% RSLogix 500 project AQUATIC CENTRE PLC UPGRADE - 21-11-05.RSS, saved by version 7.00.00.19 %
PROJECT "AQUATIC"    % processor: MicroLogix 1500 %

PROGRAM FILES
  LAD 2 "MAIN"  6 rungs
  LAD 3 "STATUS"  10 rungs
  LAD 4 "ALARMS"  24 rungs
  LAD 5 "SCREEN"  6 rungs

DATA FILES
  O0 OUTPUT  4 elements
  I1 INPUT  6 elements
  S2 STATUS  66 elements
  B3 BINARY  10 elements
  T4 TIMER  21 elements
  C5 COUNTER  1 elements
  R6 CONTROL  1 elements
  N7 INTEGER  32 elements
  F8 FLOAT  1 elements

LADDER 2 "MAIN"
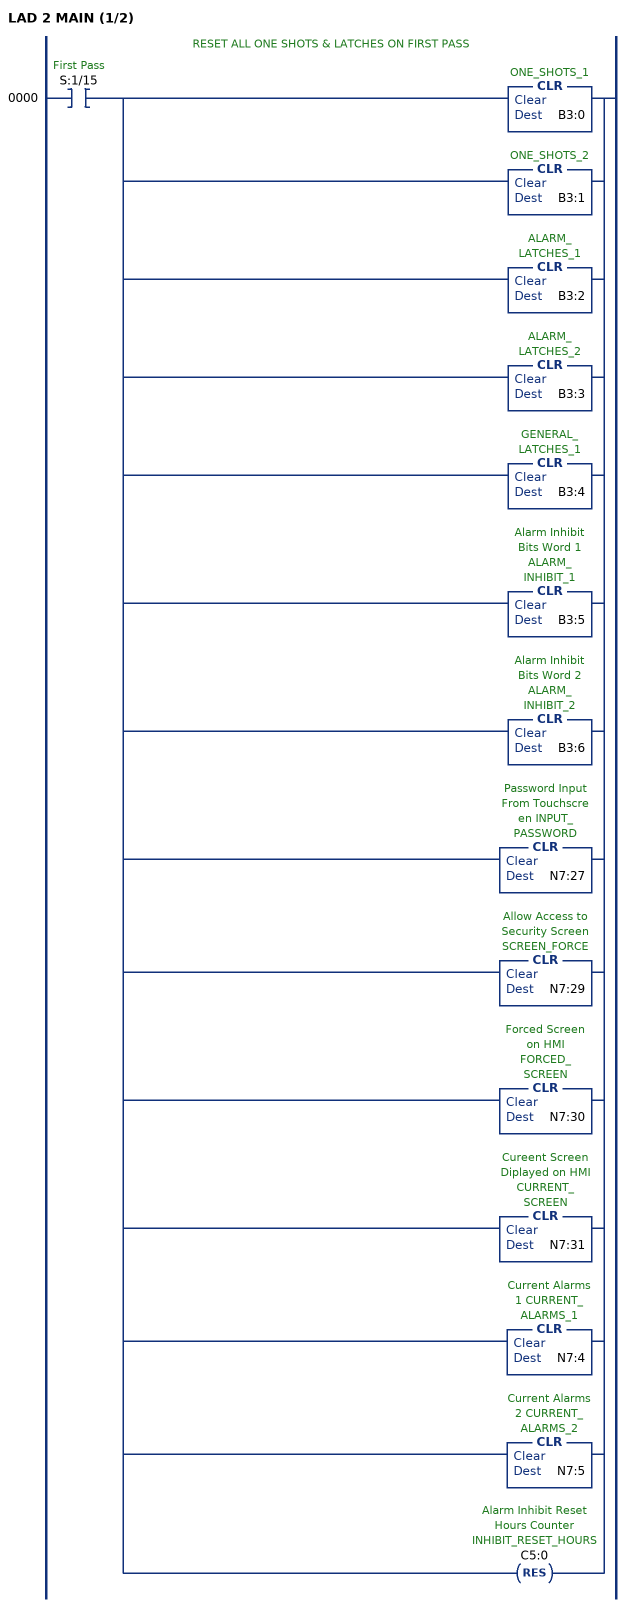
% Rung: 0 %
% RESET ALL ONE SHOTS & LATCHES ON FIRST PASS %
SOR XIC S:1/15 BST CLR B3:0 NXB CLR B3:1 NXB CLR B3:2 NXB CLR B3:3 NXB CLR B3:4 NXB CLR B3:5 NXB CLR B3:6 NXB CLR N7:27 NXB CLR N7:29 NXB CLR N7:30 NXB CLR N7:31 NXB CLR N7:4 NXB CLR N7:5 NXB RES C5:0 BND EOR
%   S:1/15  "First Pass" %
%   B3:0  ONE_SHOTS_1 %
%   B3:1  ONE_SHOTS_2 %
%   B3:2  ALARM_LATCHES_1 %
%   B3:3  ALARM_LATCHES_2 %
%   B3:4  GENERAL_LATCHES_1 %
%   B3:5  ALARM_INHIBIT_1  "Alarm Inhibit Bits Word 1" %
%   B3:6  ALARM_INHIBIT_2  "Alarm Inhibit Bits Word 2" %
%   N7:27  INPUT_PASSWORD  "Password Input From Touchscreen" %
%   N7:29  SCREEN_FORCE  "Allow Access to Security Screen" %
%   N7:30  FORCED_SCREEN  "Forced Screen on HMI" %
%   N7:31  CURRENT_SCREEN  "Cureent Screen Diplayed on HMI" %
%   N7:4  CURRENT_ALARMS_1  "Current Alarms 1" %
%   N7:5  CURRENT_ALARMS_2  "Current Alarms 2" %
%   C5:0  INHIBIT_RESET_HOURS  "Alarm Inhibit Reset Hours Counter" %

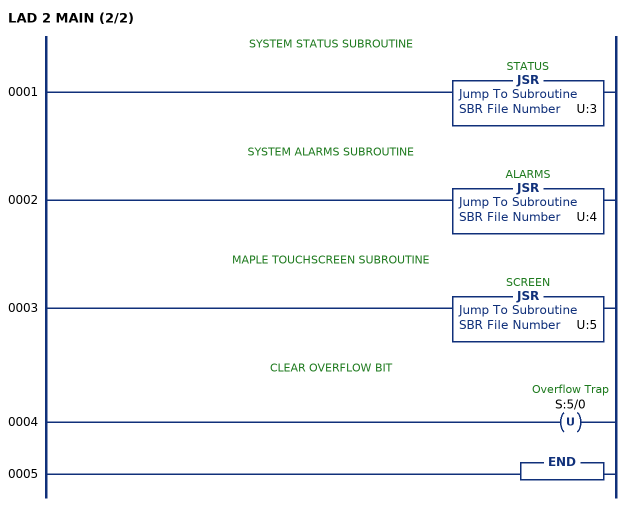
% Rung: 1 %
% SYSTEM STATUS SUBROUTINE %
SOR JSR U:3 EOR
%   U:3  STATUS %
% Rung: 2 %
% SYSTEM ALARMS SUBROUTINE %
SOR JSR U:4 EOR
%   U:4  ALARMS %
% Rung: 3 %
% MAPLE TOUCHSCREEN SUBROUTINE %
SOR JSR U:5 EOR
%   U:5  SCREEN %
% Rung: 4 %
% CLEAR OVERFLOW BIT %
SOR OTU S:5/0 EOR
%   S:5/0  "Overflow Trap" %
% Rung: 5 %
SOR END EOR

LADDER 3 "STATUS"
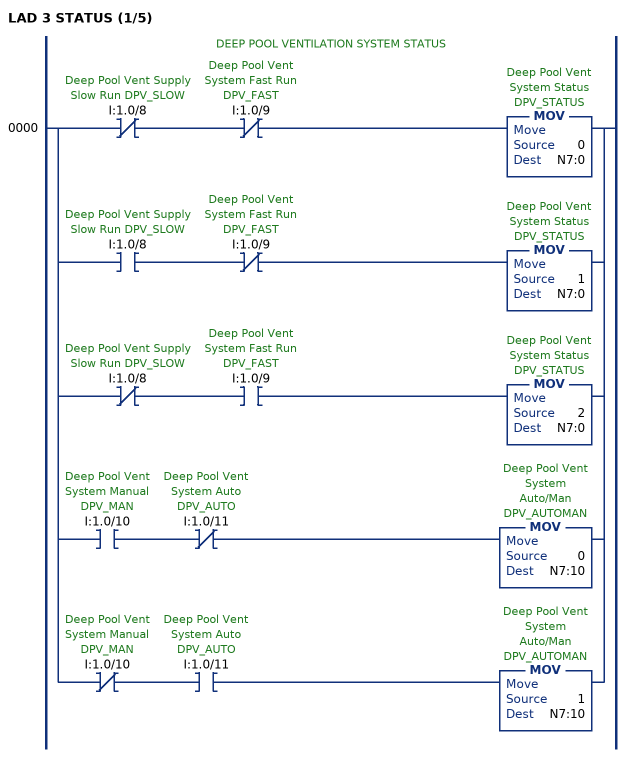
% Rung: 0 %
% DEEP POOL VENTILATION SYSTEM STATUS %
SOR BST XIO I:1.0/8 XIO I:1.0/9 MOV 0 N7:0 NXB XIC I:1.0/8 XIO I:1.0/9 MOV 1 N7:0 NXB XIO I:1.0/8 XIC I:1.0/9 MOV 2 N7:0 NXB XIC I:1.0/10 XIO I:1.0/11 MOV 0 N7:10 NXB XIO I:1.0/10 XIC I:1.0/11 MOV 1 N7:10 BND EOR
%   I:1.0/8  DPV_SLOW  "Deep Pool Vent Supply Slow Run" %
%   I:1.0/9  DPV_FAST  "Deep Pool Vent System Fast Run" %
%   N7:0  DPV_STATUS  "Deep Pool Vent System Status" %
%   I:1.0/10  DPV_MAN  "Deep Pool Vent System Manual" %
%   I:1.0/11  DPV_AUTO  "Deep Pool Vent System Auto" %
%   N7:10  DPV_AUTOMAN  "Deep Pool Vent System Auto/Man" %

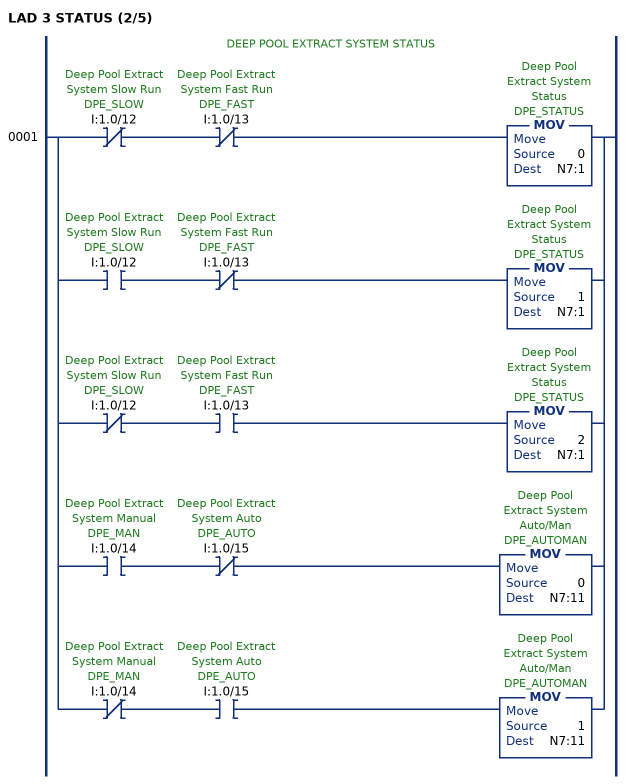
% Rung: 1 %
% DEEP POOL EXTRACT SYSTEM STATUS %
SOR BST XIO I:1.0/12 XIO I:1.0/13 MOV 0 N7:1 NXB XIC I:1.0/12 XIO I:1.0/13 MOV 1 N7:1 NXB XIO I:1.0/12 XIC I:1.0/13 MOV 2 N7:1 NXB XIC I:1.0/14 XIO I:1.0/15 MOV 0 N7:11 NXB XIO I:1.0/14 XIC I:1.0/15 MOV 1 N7:11 BND EOR
%   I:1.0/12  DPE_SLOW  "Deep Pool Extract System Slow Run" %
%   I:1.0/13  DPE_FAST  "Deep Pool Extract System Fast Run" %
%   N7:1  DPE_STATUS  "Deep Pool Extract System Status" %
%   I:1.0/14  DPE_MAN  "Deep Pool Extract System Manual" %
%   I:1.0/15  DPE_AUTO  "Deep Pool Extract System Auto" %
%   N7:11  DPE_AUTOMAN  "Deep Pool Extract System Auto/Man" %

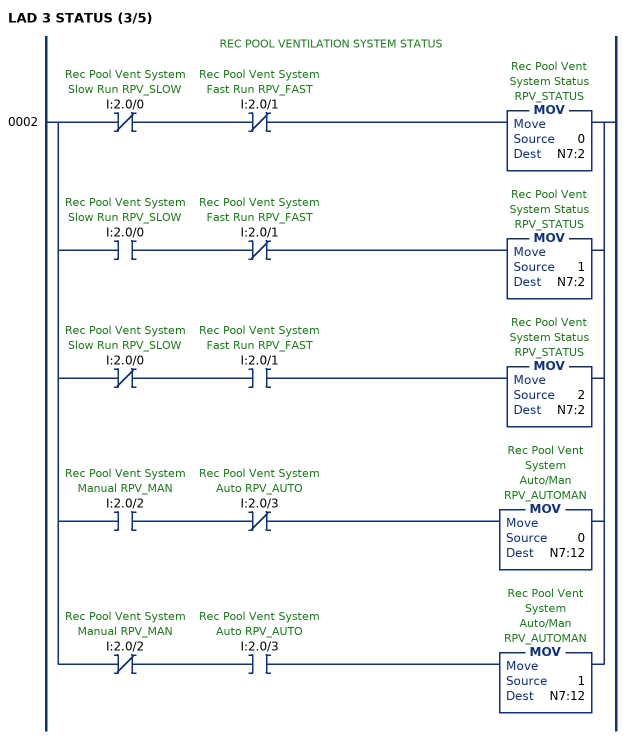
% Rung: 2 %
% REC POOL VENTILATION SYSTEM STATUS %
SOR BST XIO I:2.0/0 XIO I:2.0/1 MOV 0 N7:2 NXB XIC I:2.0/0 XIO I:2.0/1 MOV 1 N7:2 NXB XIO I:2.0/0 XIC I:2.0/1 MOV 2 N7:2 NXB XIC I:2.0/2 XIO I:2.0/3 MOV 0 N7:12 NXB XIO I:2.0/2 XIC I:2.0/3 MOV 1 N7:12 BND EOR
%   I:2.0/0  RPV_SLOW  "Rec Pool Vent System Slow Run" %
%   I:2.0/1  RPV_FAST  "Rec Pool Vent System Fast Run" %
%   N7:2  RPV_STATUS  "Rec Pool Vent System Status" %
%   I:2.0/2  RPV_MAN  "Rec Pool Vent System Manual" %
%   I:2.0/3  RPV_AUTO  "Rec Pool Vent System Auto" %
%   N7:12  RPV_AUTOMAN  "Rec Pool Vent System Auto/Man" %

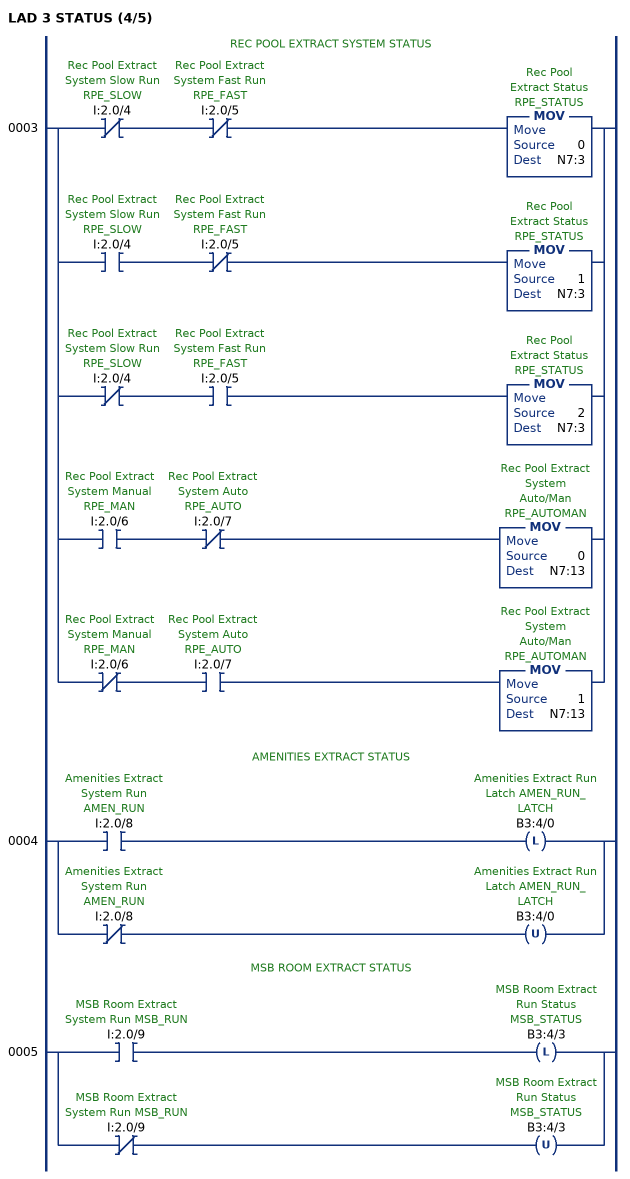
% Rung: 3 %
% REC POOL EXTRACT SYSTEM STATUS %
SOR BST XIO I:2.0/4 XIO I:2.0/5 MOV 0 N7:3 NXB XIC I:2.0/4 XIO I:2.0/5 MOV 1 N7:3 NXB XIO I:2.0/4 XIC I:2.0/5 MOV 2 N7:3 NXB XIC I:2.0/6 XIO I:2.0/7 MOV 0 N7:13 NXB XIO I:2.0/6 XIC I:2.0/7 MOV 1 N7:13 BND EOR
%   I:2.0/4  RPE_SLOW  "Rec Pool Extract System Slow Run" %
%   I:2.0/5  RPE_FAST  "Rec Pool Extract System Fast Run" %
%   N7:3  RPE_STATUS  "Rec Pool Extract Status" %
%   I:2.0/6  RPE_MAN  "Rec Pool Extract System Manual" %
%   I:2.0/7  RPE_AUTO  "Rec Pool Extract System Auto" %
%   N7:13  RPE_AUTOMAN  "Rec Pool Extract System Auto/Man" %
% Rung: 4 %
% AMENITIES EXTRACT STATUS %
SOR BST XIC I:2.0/8 OTL B3:4/0 NXB XIO I:2.0/8 OTU B3:4/0 BND EOR
%   I:2.0/8  AMEN_RUN  "Amenities Extract System Run" %
%   B3:4/0  AMEN_RUN_LATCH  "Amenities Extract Run Latch" %
% Rung: 5 %
% MSB ROOM EXTRACT STATUS %
SOR BST XIC I:2.0/9 OTL B3:4/3 NXB XIO I:2.0/9 OTU B3:4/3 BND EOR
%   I:2.0/9  MSB_RUN  "MSB Room Extract System Run" %
%   B3:4/3  MSB_STATUS  "MSB Room Extract Run Status" %

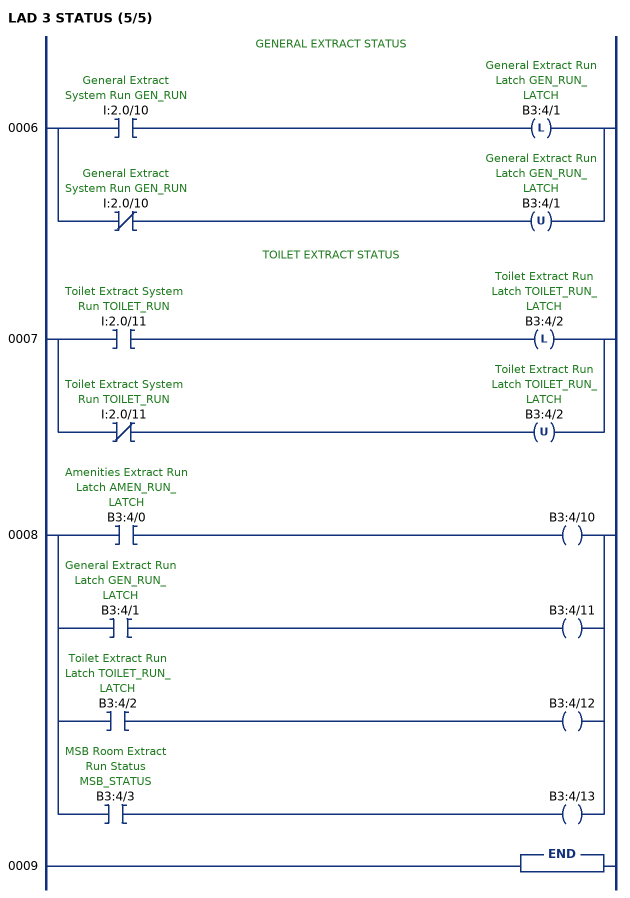
% Rung: 6 %
% GENERAL EXTRACT STATUS %
SOR BST XIC I:2.0/10 OTL B3:4/1 NXB XIO I:2.0/10 OTU B3:4/1 BND EOR
%   I:2.0/10  GEN_RUN  "General Extract System Run" %
%   B3:4/1  GEN_RUN_LATCH  "General Extract Run Latch" %
% Rung: 7 %
% TOILET EXTRACT STATUS %
SOR BST XIC I:2.0/11 OTL B3:4/2 NXB XIO I:2.0/11 OTU B3:4/2 BND EOR
%   I:2.0/11  TOILET_RUN  "Toilet Extract System Run" %
%   B3:4/2  TOILET_RUN_LATCH  "Toilet Extract Run Latch" %
% Rung: 8 %
SOR BST XIC B3:4/0 OTE B3:4/10 NXB XIC B3:4/1 OTE B3:4/11 NXB XIC B3:4/2 OTE B3:4/12 NXB XIC B3:4/3 OTE B3:4/13 BND EOR
%   B3:4/0  AMEN_RUN_LATCH  "Amenities Extract Run Latch" %
%   B3:4/1  GEN_RUN_LATCH  "General Extract Run Latch" %
%   B3:4/2  TOILET_RUN_LATCH  "Toilet Extract Run Latch" %
%   B3:4/3  MSB_STATUS  "MSB Room Extract Run Status" %
% Rung: 9 %
SOR END EOR

LADDER 4 "ALARMS"
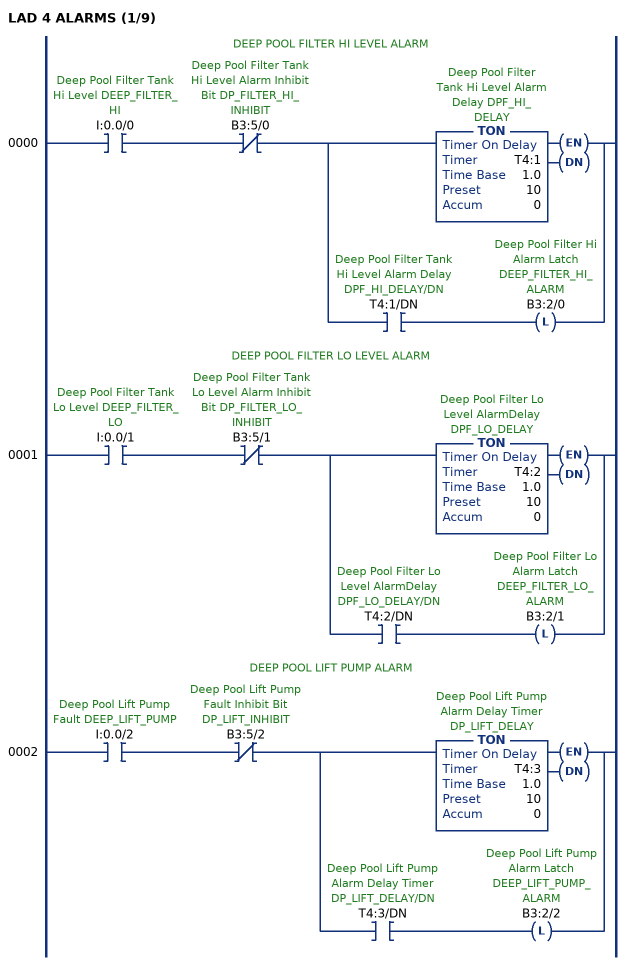
% Rung: 0 %
% DEEP POOL FILTER HI LEVEL ALARM %
SOR XIC I:0.0/0 XIO B3:5/0 BST TON T4:1 1.0 10 0 NXB XIC T4:1/DN OTL B3:2/0 BND EOR
%   I:0.0/0  DEEP_FILTER_HI  "Deep Pool Filter Tank Hi Level" %
%   B3:5/0  DP_FILTER_HI_INHIBIT  "Deep Pool Filter Tank Hi Level Alarm Inhibit Bit" %
%   T4:1  DPF_HI_DELAY  "Deep Pool Filter Tank Hi Level Alarm Delay" %
%   B3:2/0  DEEP_FILTER_HI_ALARM  "Deep Pool Filter Hi Alarm Latch" %
% Rung: 1 %
% DEEP POOL FILTER LO LEVEL ALARM %
SOR XIC I:0.0/1 XIO B3:5/1 BST TON T4:2 1.0 10 0 NXB XIC T4:2/DN OTL B3:2/1 BND EOR
%   I:0.0/1  DEEP_FILTER_LO  "Deep Pool Filter Tank Lo Level" %
%   B3:5/1  DP_FILTER_LO_INHIBIT  "Deep Pool Filter Tank Lo Level Alarm Inhibit Bit" %
%   T4:2  DPF_LO_DELAY  "Deep Pool Filter Lo Level AlarmDelay" %
%   B3:2/1  DEEP_FILTER_LO_ALARM  "Deep Pool Filter Lo Alarm Latch" %
% Rung: 2 %
% DEEP POOL LIFT PUMP ALARM %
SOR XIC I:0.0/2 XIO B3:5/2 BST TON T4:3 1.0 10 0 NXB XIC T4:3/DN OTL B3:2/2 BND EOR
%   I:0.0/2  DEEP_LIFT_PUMP  "Deep Pool Lift Pump Fault" %
%   B3:5/2  DP_LIFT_INHIBIT  "Deep Pool Lift Pump Fault Inhibit Bit" %
%   T4:3  DP_LIFT_DELAY  "Deep Pool Lift Pump Alarm Delay Timer" %
%   B3:2/2  DEEP_LIFT_PUMP_ALARM  "Deep Pool Lift Pump Alarm Latch" %

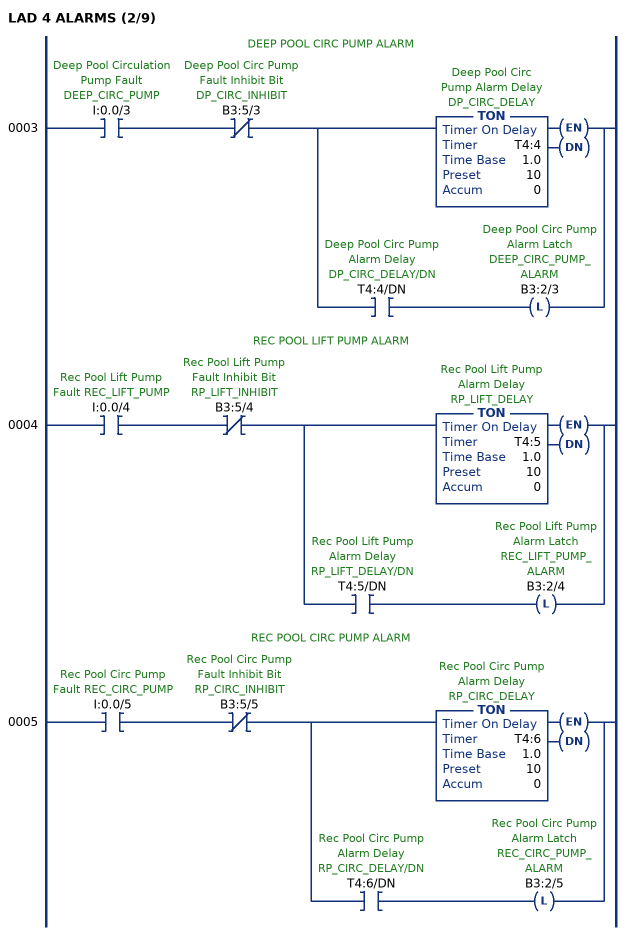
% Rung: 3 %
% DEEP POOL CIRC PUMP ALARM %
SOR XIC I:0.0/3 XIO B3:5/3 BST TON T4:4 1.0 10 0 NXB XIC T4:4/DN OTL B3:2/3 BND EOR
%   I:0.0/3  DEEP_CIRC_PUMP  "Deep Pool Circulation Pump Fault" %
%   B3:5/3  DP_CIRC_INHIBIT  "Deep Pool Circ Pump Fault Inhibit Bit" %
%   T4:4  DP_CIRC_DELAY  "Deep Pool Circ Pump Alarm Delay" %
%   B3:2/3  DEEP_CIRC_PUMP_ALARM  "Deep Pool Circ Pump Alarm Latch" %
% Rung: 4 %
% REC POOL LIFT PUMP ALARM %
SOR XIC I:0.0/4 XIO B3:5/4 BST TON T4:5 1.0 10 0 NXB XIC T4:5/DN OTL B3:2/4 BND EOR
%   I:0.0/4  REC_LIFT_PUMP  "Rec Pool Lift Pump Fault" %
%   B3:5/4  RP_LIFT_INHIBIT  "Rec Pool Lift Pump Fault Inhibit Bit" %
%   T4:5  RP_LIFT_DELAY  "Rec Pool Lift Pump Alarm Delay" %
%   B3:2/4  REC_LIFT_PUMP_ALARM  "Rec Pool Lift Pump Alarm Latch" %
% Rung: 5 %
% REC POOL CIRC PUMP ALARM %
SOR XIC I:0.0/5 XIO B3:5/5 BST TON T4:6 1.0 10 0 NXB XIC T4:6/DN OTL B3:2/5 BND EOR
%   I:0.0/5  REC_CIRC_PUMP  "Rec Pool Circ Pump Fault" %
%   B3:5/5  RP_CIRC_INHIBIT  "Rec Pool Circ Pump Fault Inhibit Bit" %
%   T4:6  RP_CIRC_DELAY  "Rec Pool Circ Pump Alarm Delay" %
%   B3:2/5  REC_CIRC_PUMP_ALARM  "Rec Pool Circ Pump Alarm Latch" %

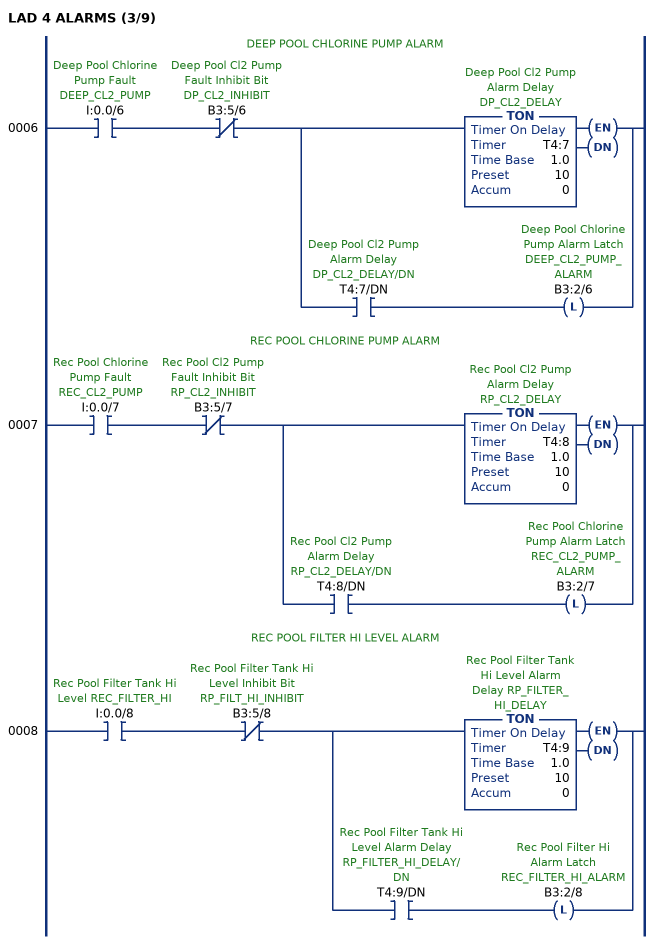
% Rung: 6 %
% DEEP POOL CHLORINE PUMP ALARM %
SOR XIC I:0.0/6 XIO B3:5/6 BST TON T4:7 1.0 10 0 NXB XIC T4:7/DN OTL B3:2/6 BND EOR
%   I:0.0/6  DEEP_CL2_PUMP  "Deep Pool Chlorine Pump Fault" %
%   B3:5/6  DP_CL2_INHIBIT  "Deep Pool Cl2 Pump Fault Inhibit Bit" %
%   T4:7  DP_CL2_DELAY  "Deep Pool Cl2 Pump Alarm Delay" %
%   B3:2/6  DEEP_CL2_PUMP_ALARM  "Deep Pool Chlorine Pump Alarm Latch" %
% Rung: 7 %
% REC POOL CHLORINE PUMP ALARM %
SOR XIC I:0.0/7 XIO B3:5/7 BST TON T4:8 1.0 10 0 NXB XIC T4:8/DN OTL B3:2/7 BND EOR
%   I:0.0/7  REC_CL2_PUMP  "Rec Pool Chlorine Pump Fault" %
%   B3:5/7  RP_CL2_INHIBIT  "Rec Pool Cl2 Pump Fault Inhibit Bit" %
%   T4:8  RP_CL2_DELAY  "Rec Pool Cl2 Pump Alarm Delay" %
%   B3:2/7  REC_CL2_PUMP_ALARM  "Rec Pool Chlorine Pump Alarm Latch" %
% Rung: 8 %
% REC POOL FILTER HI LEVEL ALARM %
SOR XIC I:0.0/8 XIO B3:5/8 BST TON T4:9 1.0 10 0 NXB XIC T4:9/DN OTL B3:2/8 BND EOR
%   I:0.0/8  REC_FILTER_HI  "Rec Pool Filter Tank Hi Level" %
%   B3:5/8  RP_FILT_HI_INHIBIT  "Rec Pool Filter Tank Hi Level Inhibit Bit" %
%   T4:9  RP_FILTER_HI_DELAY  "Rec Pool Filter Tank Hi Level Alarm Delay" %
%   B3:2/8  REC_FILTER_HI_ALARM  "Rec Pool Filter Hi Alarm Latch" %

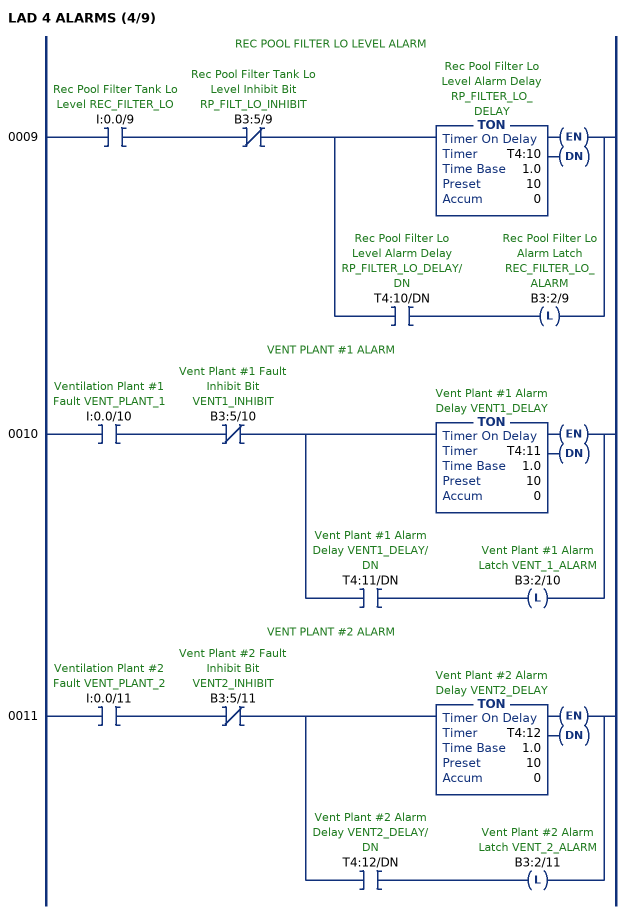
% Rung: 9 %
% REC POOL FILTER LO LEVEL ALARM %
SOR XIC I:0.0/9 XIO B3:5/9 BST TON T4:10 1.0 10 0 NXB XIC T4:10/DN OTL B3:2/9 BND EOR
%   I:0.0/9  REC_FILTER_LO  "Rec Pool Filter Tank Lo Level" %
%   B3:5/9  RP_FILT_LO_INHIBIT  "Rec Pool Filter Tank Lo Level Inhibit Bit" %
%   T4:10  RP_FILTER_LO_DELAY  "Rec Pool Filter Lo Level Alarm Delay" %
%   B3:2/9  REC_FILTER_LO_ALARM  "Rec Pool Filter Lo Alarm Latch" %
% Rung: 10 %
% VENT PLANT #1 ALARM %
SOR XIC I:0.0/10 XIO B3:5/10 BST TON T4:11 1.0 10 0 NXB XIC T4:11/DN OTL B3:2/10 BND EOR
%   I:0.0/10  VENT_PLANT_1  "Ventilation Plant #1 Fault" %
%   B3:5/10  VENT1_INHIBIT  "Vent Plant #1 Fault Inhibit Bit" %
%   T4:11  VENT1_DELAY  "Vent Plant #1 Alarm Delay" %
%   B3:2/10  VENT_1_ALARM  "Vent Plant #1 Alarm Latch" %
% Rung: 11 %
% VENT PLANT #2 ALARM %
SOR XIC I:0.0/11 XIO B3:5/11 BST TON T4:12 1.0 10 0 NXB XIC T4:12/DN OTL B3:2/11 BND EOR
%   I:0.0/11  VENT_PLANT_2  "Ventilation Plant #2 Fault" %
%   B3:5/11  VENT2_INHIBIT  "Vent Plant #2 Fault Inhibit Bit" %
%   T4:12  VENT2_DELAY  "Vent Plant #2 Alarm Delay" %
%   B3:2/11  VENT_2_ALARM  "Vent Plant #2 Alarm Latch" %

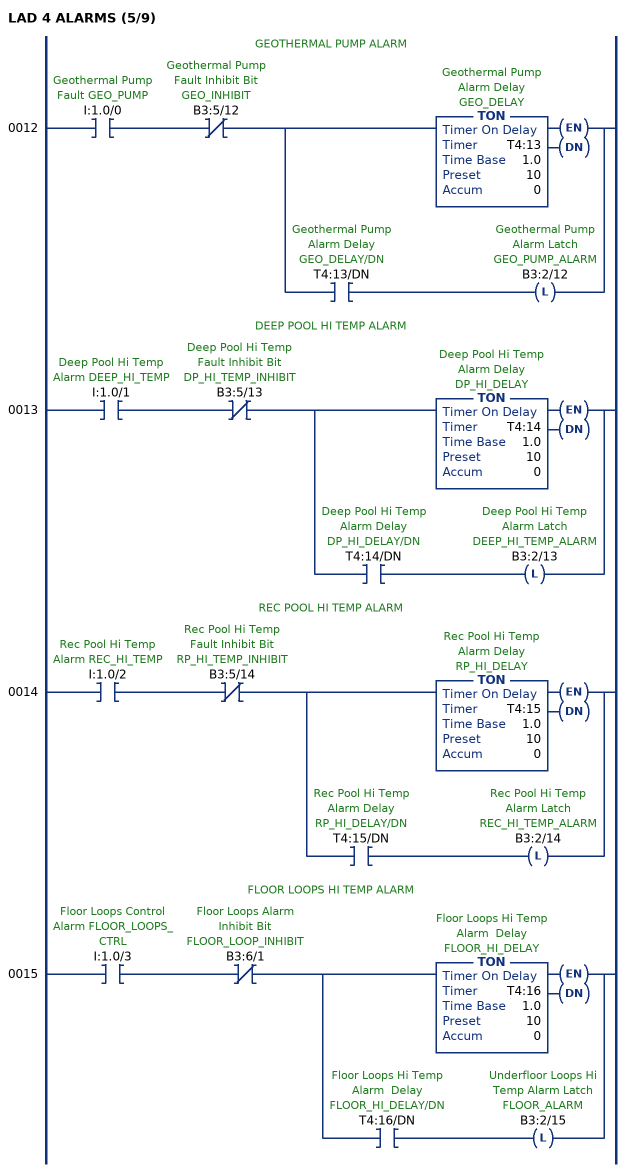
% Rung: 12 %
% GEOTHERMAL PUMP ALARM %
SOR XIC I:1.0/0 XIO B3:5/12 BST TON T4:13 1.0 10 0 NXB XIC T4:13/DN OTL B3:2/12 BND EOR
%   I:1.0/0  GEO_PUMP  "Geothermal Pump Fault" %
%   B3:5/12  GEO_INHIBIT  "Geothermal Pump Fault Inhibit Bit" %
%   T4:13  GEO_DELAY  "Geothermal Pump Alarm Delay" %
%   B3:2/12  GEO_PUMP_ALARM  "Geothermal Pump Alarm Latch" %
% Rung: 13 %
% DEEP POOL HI TEMP ALARM %
SOR XIC I:1.0/1 XIO B3:5/13 BST TON T4:14 1.0 10 0 NXB XIC T4:14/DN OTL B3:2/13 BND EOR
%   I:1.0/1  DEEP_HI_TEMP  "Deep Pool Hi Temp Alarm" %
%   B3:5/13  DP_HI_TEMP_INHIBIT  "Deep Pool Hi Temp Fault Inhibit Bit" %
%   T4:14  DP_HI_DELAY  "Deep Pool Hi Temp Alarm Delay" %
%   B3:2/13  DEEP_HI_TEMP_ALARM  "Deep Pool Hi Temp Alarm Latch" %
% Rung: 14 %
% REC POOL HI TEMP ALARM %
SOR XIC I:1.0/2 XIO B3:5/14 BST TON T4:15 1.0 10 0 NXB XIC T4:15/DN OTL B3:2/14 BND EOR
%   I:1.0/2  REC_HI_TEMP  "Rec Pool Hi Temp Alarm" %
%   B3:5/14  RP_HI_TEMP_INHIBIT  "Rec Pool Hi Temp Fault Inhibit Bit" %
%   T4:15  RP_HI_DELAY  "Rec Pool Hi Temp Alarm Delay" %
%   B3:2/14  REC_HI_TEMP_ALARM  "Rec Pool Hi Temp Alarm Latch" %
% Rung: 15 %
% FLOOR LOOPS HI TEMP ALARM %
SOR XIC I:1.0/3 XIO B3:6/1 BST TON T4:16 1.0 10 0 NXB XIC T4:16/DN OTL B3:2/15 BND EOR
%   I:1.0/3  FLOOR_LOOPS_CTRL  "Floor Loops Control Alarm" %
%   B3:6/1  FLOOR_LOOP_INHIBIT  "Floor Loops Alarm Inhibit Bit" %
%   T4:16  FLOOR_HI_DELAY  "Floor Loops Hi Temp Alarm  Delay" %
%   B3:2/15  FLOOR_ALARM  "Underfloor Loops Hi Temp Alarm Latch" %

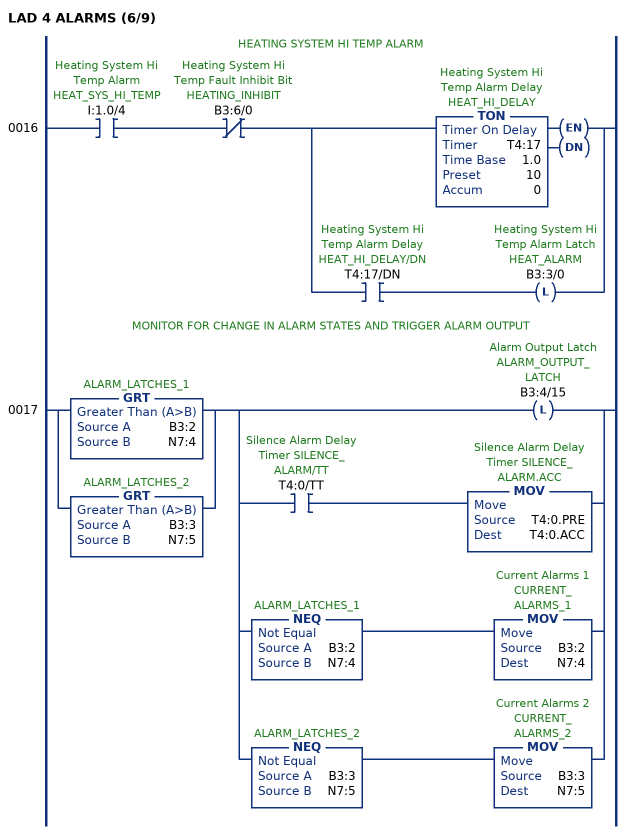
% Rung: 16 %
% HEATING SYSTEM HI TEMP ALARM %
SOR XIC I:1.0/4 XIO B3:6/0 BST TON T4:17 1.0 10 0 NXB XIC T4:17/DN OTL B3:3/0 BND EOR
%   I:1.0/4  HEAT_SYS_HI_TEMP  "Heating System Hi Temp Alarm" %
%   B3:6/0  HEATING_INHIBIT  "Heating System Hi Temp Fault Inhibit Bit" %
%   T4:17  HEAT_HI_DELAY  "Heating System Hi Temp Alarm Delay" %
%   B3:3/0  HEAT_ALARM  "Heating System Hi Temp Alarm Latch" %
% Rung: 17 %
% MONITOR FOR CHANGE IN ALARM STATES AND TRIGGER ALARM OUTPUT %
SOR BST GRT B3:2 N7:4 NXB GRT B3:3 N7:5 BND BST OTL B3:4/15 NXB XIC T4:0/TT MOV T4:0.PRE T4:0.ACC NXB NEQ B3:2 N7:4 MOV B3:2 N7:4 NXB NEQ B3:3 N7:5 MOV B3:3 N7:5 BND EOR
%   B3:2  ALARM_LATCHES_1 %
%   N7:4  CURRENT_ALARMS_1  "Current Alarms 1" %
%   B3:3  ALARM_LATCHES_2 %
%   N7:5  CURRENT_ALARMS_2  "Current Alarms 2" %
%   B3:4/15  ALARM_OUTPUT_LATCH  "Alarm Output Latch" %
%   T4:0  SILENCE_ALARM  "Silence Alarm Delay Timer" %

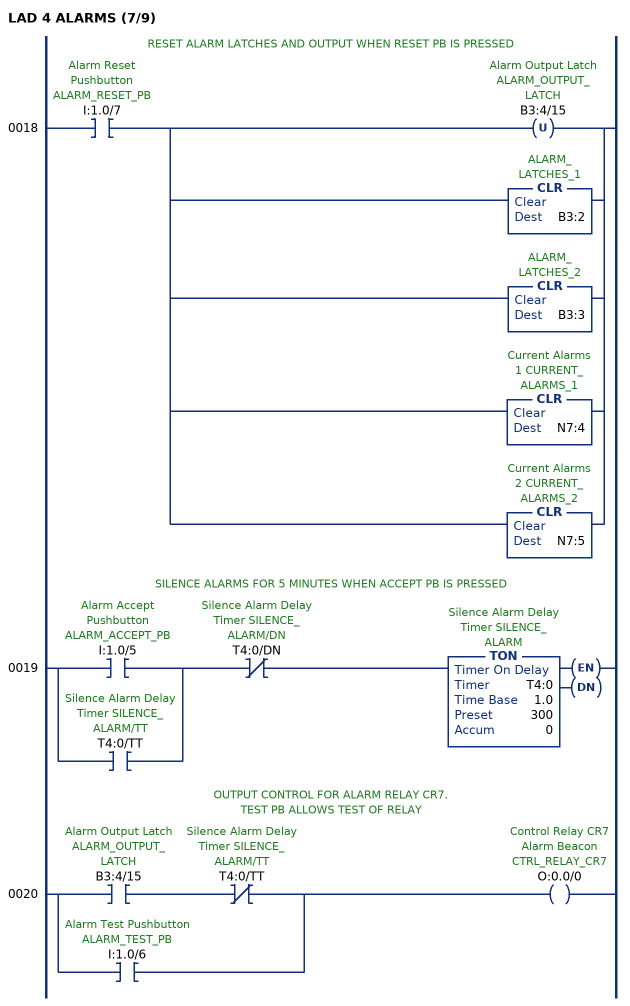
% Rung: 18 %
% RESET ALARM LATCHES AND OUTPUT WHEN RESET PB IS PRESSED %
SOR XIC I:1.0/7 BST OTU B3:4/15 NXB CLR B3:2 NXB CLR B3:3 NXB CLR N7:4 NXB CLR N7:5 BND EOR
%   I:1.0/7  ALARM_RESET_PB  "Alarm Reset Pushbutton" %
%   B3:4/15  ALARM_OUTPUT_LATCH  "Alarm Output Latch" %
%   B3:2  ALARM_LATCHES_1 %
%   B3:3  ALARM_LATCHES_2 %
%   N7:4  CURRENT_ALARMS_1  "Current Alarms 1" %
%   N7:5  CURRENT_ALARMS_2  "Current Alarms 2" %
% Rung: 19 %
% SILENCE ALARMS FOR 5 MINUTES WHEN ACCEPT PB IS PRESSED %
SOR BST XIC I:1.0/5 NXB XIC T4:0/TT BND XIO T4:0/DN TON T4:0 1.0 300 0 EOR
%   I:1.0/5  ALARM_ACCEPT_PB  "Alarm Accept Pushbutton" %
%   T4:0  SILENCE_ALARM  "Silence Alarm Delay Timer" %
% Rung: 20 %
% OUTPUT CONTROL FOR ALARM RELAY CR7.
% TEST PB ALLOWS TEST OF RELAY %
SOR BST XIC B3:4/15 XIO T4:0/TT NXB XIC I:1.0/6 BND OTE O:0.0/0 EOR
%   B3:4/15  ALARM_OUTPUT_LATCH  "Alarm Output Latch" %
%   T4:0  SILENCE_ALARM  "Silence Alarm Delay Timer" %
%   I:1.0/6  ALARM_TEST_PB  "Alarm Test Pushbutton" %
%   O:0.0/0  CTRL_RELAY_CR7  "Control Relay CR7 Alarm Beacon" %

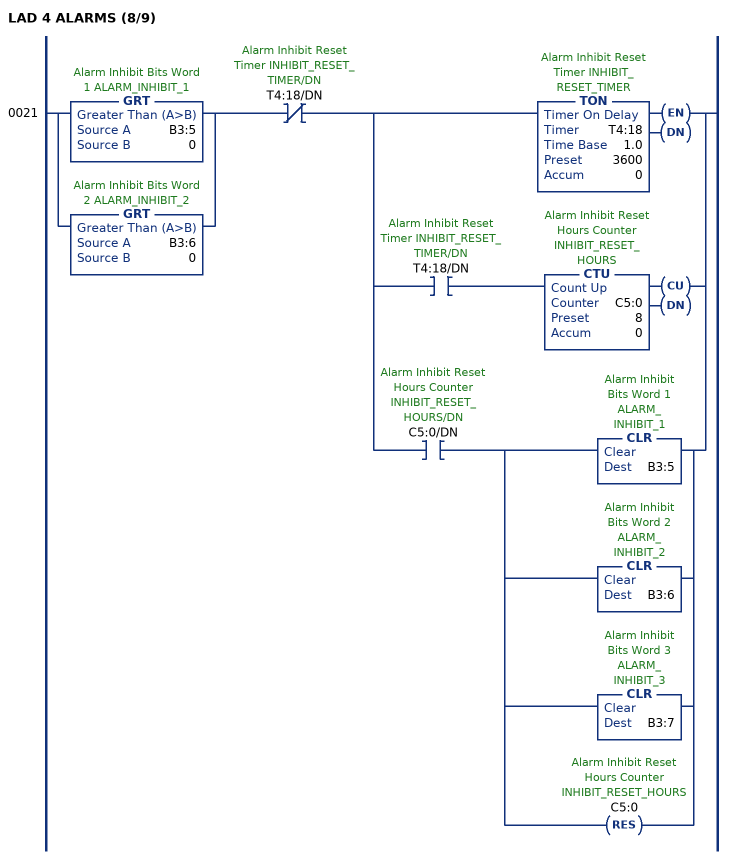
% Rung: 21 %
SOR BST GRT B3:5 0 NXB GRT B3:6 0 BND XIO T4:18/DN BST TON T4:18 1.0 3600 0 NXB XIC T4:18/DN CTU C5:0 8 0 NXB XIC C5:0/DN BST CLR B3:5 NXB CLR B3:6 NXB CLR B3:7 NXB RES C5:0 BND BND EOR
%   B3:5  ALARM_INHIBIT_1  "Alarm Inhibit Bits Word 1" %
%   B3:6  ALARM_INHIBIT_2  "Alarm Inhibit Bits Word 2" %
%   T4:18  INHIBIT_RESET_TIMER  "Alarm Inhibit Reset Timer" %
%   C5:0  INHIBIT_RESET_HOURS  "Alarm Inhibit Reset Hours Counter" %
%   B3:7  ALARM_INHIBIT_3  "Alarm Inhibit Bits Word 3" %

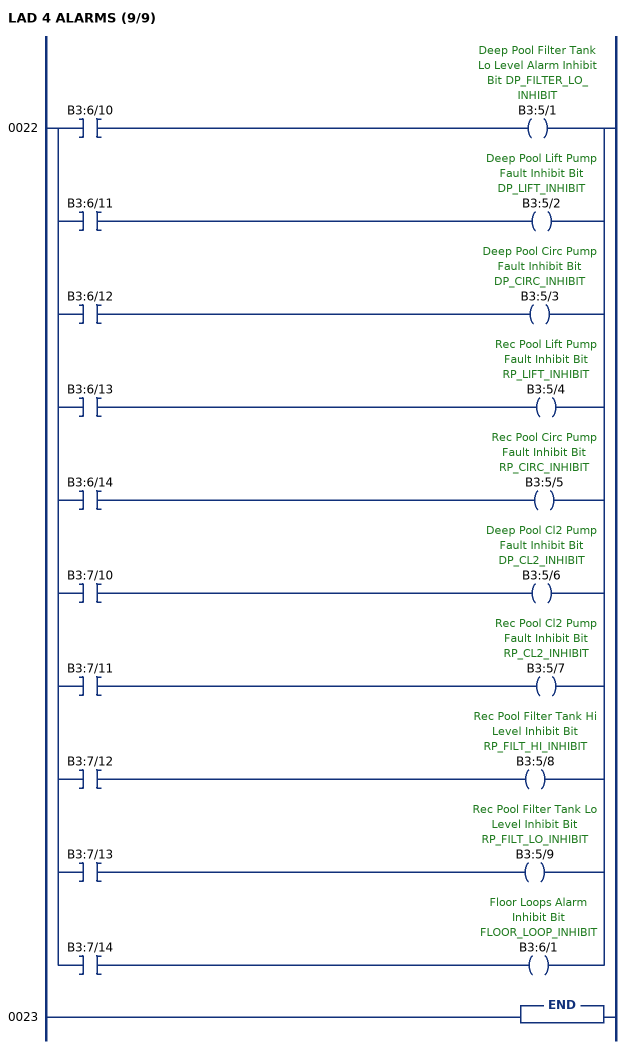
% Rung: 22 %
SOR BST XIC B3:6/10 OTE B3:5/1 NXB XIC B3:6/11 OTE B3:5/2 NXB XIC B3:6/12 OTE B3:5/3 NXB XIC B3:6/13 OTE B3:5/4 NXB XIC B3:6/14 OTE B3:5/5 NXB XIC B3:7/10 OTE B3:5/6 NXB XIC B3:7/11 OTE B3:5/7 NXB XIC B3:7/12 OTE B3:5/8 NXB XIC B3:7/13 OTE B3:5/9 NXB XIC B3:7/14 OTE B3:6/1 BND EOR
%   B3:5/1  DP_FILTER_LO_INHIBIT  "Deep Pool Filter Tank Lo Level Alarm Inhibit Bit" %
%   B3:5/2  DP_LIFT_INHIBIT  "Deep Pool Lift Pump Fault Inhibit Bit" %
%   B3:5/3  DP_CIRC_INHIBIT  "Deep Pool Circ Pump Fault Inhibit Bit" %
%   B3:5/4  RP_LIFT_INHIBIT  "Rec Pool Lift Pump Fault Inhibit Bit" %
%   B3:5/5  RP_CIRC_INHIBIT  "Rec Pool Circ Pump Fault Inhibit Bit" %
%   B3:5/6  DP_CL2_INHIBIT  "Deep Pool Cl2 Pump Fault Inhibit Bit" %
%   B3:5/7  RP_CL2_INHIBIT  "Rec Pool Cl2 Pump Fault Inhibit Bit" %
%   B3:5/8  RP_FILT_HI_INHIBIT  "Rec Pool Filter Tank Hi Level Inhibit Bit" %
%   B3:5/9  RP_FILT_LO_INHIBIT  "Rec Pool Filter Tank Lo Level Inhibit Bit" %
%   B3:6/1  FLOOR_LOOP_INHIBIT  "Floor Loops Alarm Inhibit Bit" %
% Rung: 23 %
SOR END EOR

LADDER 5 "SCREEN"
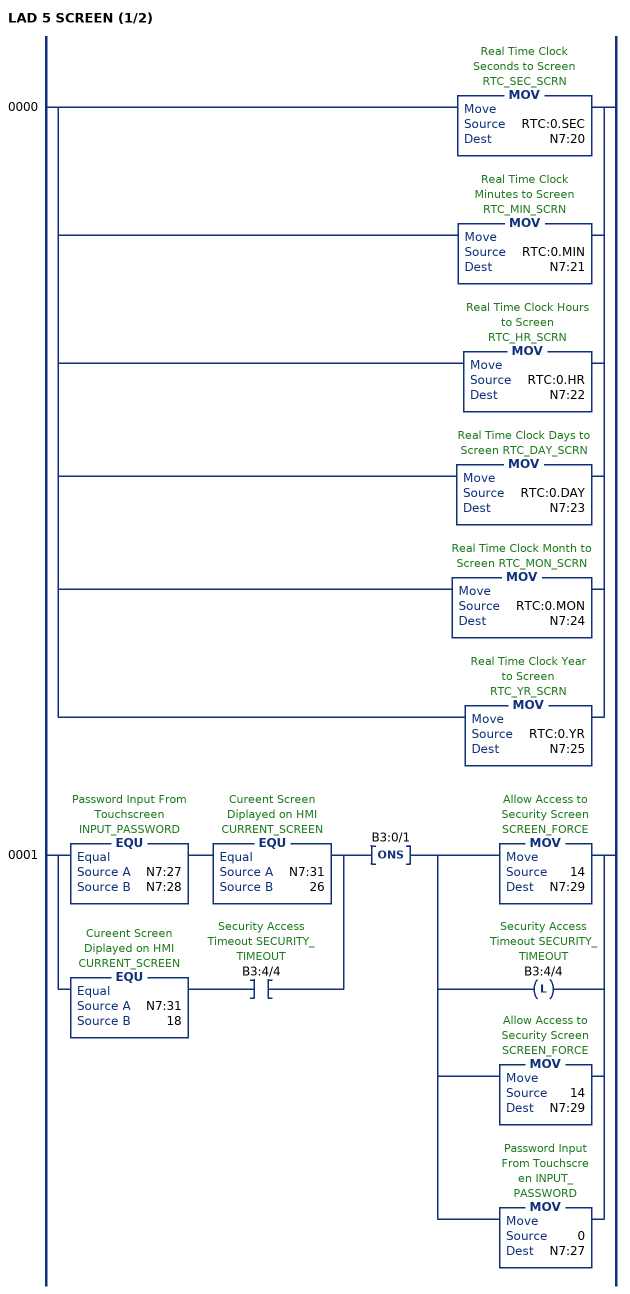
% Rung: 0 %
SOR BST MOV RTC:0.SEC N7:20 NXB MOV RTC:0.MIN N7:21 NXB MOV RTC:0.HR N7:22 NXB MOV RTC:0.DAY N7:23 NXB MOV RTC:0.MON N7:24 NXB MOV RTC:0.YR N7:25 BND EOR
%   RTC:0.SEC  RTC_SEC  "Real Time Clock Seconds" %
%   N7:20  RTC_SEC_SCRN  "Real Time Clock Seconds to Screen" %
%   N7:21  RTC_MIN_SCRN  "Real Time Clock Minutes to Screen" %
%   N7:22  RTC_HR_SCRN  "Real Time Clock Hours to Screen" %
%   N7:23  RTC_DAY_SCRN  "Real Time Clock Days to Screen" %
%   N7:24  RTC_MON_SCRN  "Real Time Clock Month to Screen" %
%   N7:25  RTC_YR_SCRN  "Real Time Clock Year to Screen" %
% Rung: 1 %
SOR BST EQU N7:27 N7:28 EQU N7:31 26 NXB EQU N7:31 18 XIC B3:4/4 BND ONS B3:0/1 BST MOV 14 N7:29 NXB OTL B3:4/4 NXB MOV 14 N7:29 NXB MOV 0 N7:27 BND EOR
%   N7:27  INPUT_PASSWORD  "Password Input From Touchscreen" %
%   N7:28  SYSTEM_PASSWORD  "Security Password" %
%   N7:31  CURRENT_SCREEN  "Cureent Screen Diplayed on HMI" %
%   B3:4/4  SECURITY_TIMEOUT  "Security Access Timeout" %
%   N7:29  SCREEN_FORCE  "Allow Access to Security Screen" %

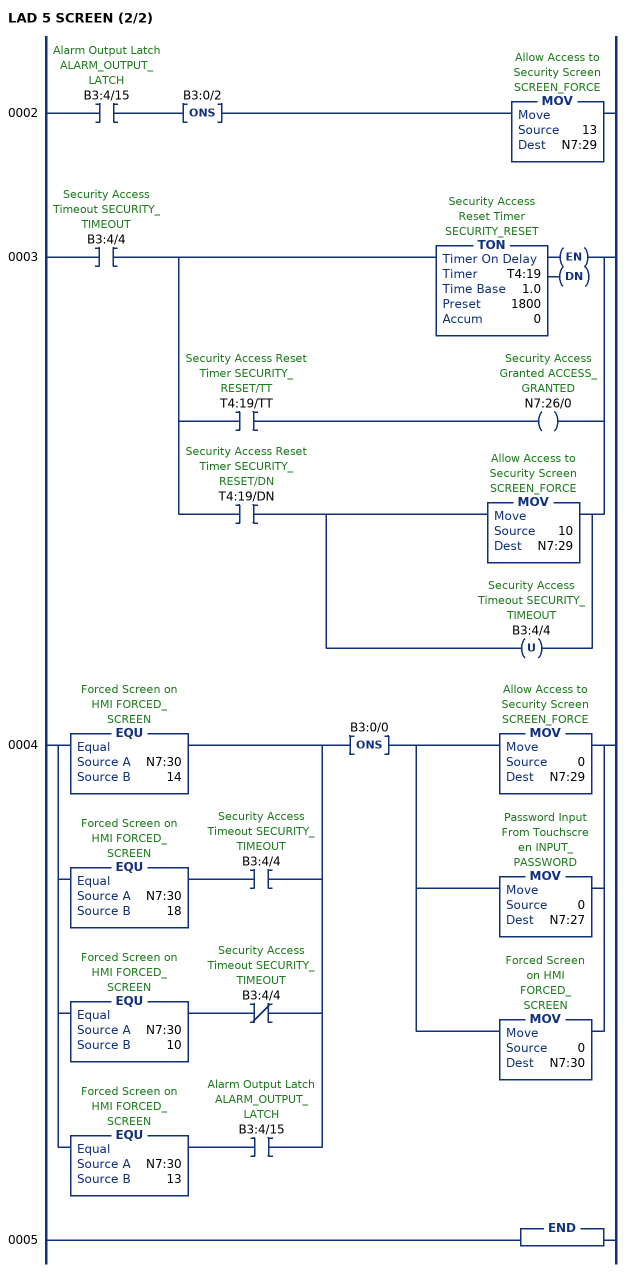
% Rung: 2 %
SOR XIC B3:4/15 ONS B3:0/2 MOV 13 N7:29 EOR
%   B3:4/15  ALARM_OUTPUT_LATCH  "Alarm Output Latch" %
%   N7:29  SCREEN_FORCE  "Allow Access to Security Screen" %
% Rung: 3 %
SOR XIC B3:4/4 BST TON T4:19 1.0 1800 0 NXB XIC T4:19/TT OTE N7:26/0 NXB XIC T4:19/DN BST MOV 10 N7:29 NXB OTU B3:4/4 BND BND EOR
%   B3:4/4  SECURITY_TIMEOUT  "Security Access Timeout" %
%   T4:19  SECURITY_RESET  "Security Access Reset Timer" %
%   N7:26/0  ACCESS_GRANTED  "Security Access Granted" %
%   N7:29  SCREEN_FORCE  "Allow Access to Security Screen" %
% Rung: 4 %
SOR BST EQU N7:30 14 NXB EQU N7:30 18 XIC B3:4/4 NXB EQU N7:30 10 XIO B3:4/4 NXB EQU N7:30 13 XIC B3:4/15 BND ONS B3:0/0 BST MOV 0 N7:29 NXB MOV 0 N7:27 NXB MOV 0 N7:30 BND EOR
%   N7:30  FORCED_SCREEN  "Forced Screen on HMI" %
%   B3:4/4  SECURITY_TIMEOUT  "Security Access Timeout" %
%   B3:4/15  ALARM_OUTPUT_LATCH  "Alarm Output Latch" %
%   N7:29  SCREEN_FORCE  "Allow Access to Security Screen" %
%   N7:27  INPUT_PASSWORD  "Password Input From Touchscreen" %
% Rung: 5 %
SOR END EOR

OTHER DOCUMENTED ADDRESSES
    "Deep Pool Filter Tank Hi Level Alarm Inhibit Bit"
  B3:8  ALARM_INHIBIT_4  "Alarm Inhibit Bits Word 4"
  N7:26  STATUS_BITS  "Status Bits to Touchscreen"
  T4:20  SECURITY_SCRN_DELAY  "Delay to change Security Screens"

COMMENTS NOT ATTACHED TO A CURRENT RUNG
  B3:4/0: AMENITIES EXTRACT STATUS

REVISION NOTES
  0: Installed January 2006

DATA TABLE (non-zero values as saved)
DATA B3
% B3:0 % 0X0000 0X0000 0X0000 0X0000 0X3C0F 0X0000 0X0000 0X0000 0X0000 0X0000
DATA T4
% .PRE .ACC %
% T4:0 % 300 0
% T4:1 % 10 0
% T4:2 % 10 0
% T4:3 % 10 0
% T4:4 % 10 0
% T4:5 % 10 0
% T4:6 % 10 0
% T4:7 % 10 0
% T4:8 % 10 0
% T4:9 % 10 0
% T4:10 % 10 0
% T4:11 % 10 0
% T4:12 % 10 0
% T4:13 % 10 0
% T4:14 % 10 0
% T4:15 % 10 0
% T4:16 % 10 0
% T4:17 % 10 0
% T4:18 % 3600 0
% T4:19 % 1800 0
% T4:20 % 50 0
DATA C5
% .PRE .ACC %
% C5:0 % 8 0
DATA N7
% N7:0 % 2 2 2 2 0 0 0 0 0 0
% N7:10 % 1 1 1 1 0 0 0 253 0 0
% N7:20 % 18 5 10 20 1 2006 0 0 1234 0
% N7:30 % 0 27
